// TIA Portal V20 export
TYPE "typeCmControlNodeInterlock"
// stored: Namespace Unit1.Em5
   STRUCT
      ngAndManualInput { ExternalWritable := 'False'} : "LER_typeAxisInterlock";
      magazine { ExternalWritable := 'False'} : "LER_typeAxisInterlock";
      ngAndManualInputCylinder { ExternalWritable := 'False'} : "LER_typeTwoWayActuatorInterlock";
      ngAndManualInputVacuum1 { ExternalWritable := 'False'} : "LER_typeTwoWayActuatorInterlock";
      ngAndManualInputVacuum2 { ExternalWritable := 'False'} : "LER_typeTwoWayActuatorInterlock";
      ngAndManualInputVibrator1 { ExternalWritable := 'False'} : "LER_typeTwoWayActuatorInterlock";
      ngAndManualInputVibrator2 { ExternalWritable := 'False'} : "LER_typeTwoWayActuatorInterlock";
      magazineLockCylinder { ExternalWritable := 'False'} : "LER_typeTwoWayActuatorInterlock";
   END_STRUCT;
END_TYPE
